# B&R Automation Studio project OPSU1
Automation Studio 4.5.2.102

## Configuration Real

### Task classes (Cpu.sw)
```
Cyclic#4:
  Main <- Main.prg
Libraries: motor
```

### Hardware
```
4PP065_0571_P74 : 4PP065.0571-P74 v1.1.2.0
  Connector IF5:
    ActivateDevice = 1
  ConfigurationID = kvbo0721lab1_Real
  Simulation = 1
```

## Logical view

Binary libraries used (declarations not repeated): operator, runtime, astime, AsIecCon

### Package Logical/Libraries - Global libraries

### Library Logical/Libraries/motor (ANSIC)

#### motor.fun - Exported functions and function blocks
```iecst
{REDUND_ERROR} {REDUND_UNREPLICABLE} FUNCTION_BLOCK FB_Motor (*TODO: Add your comment here*) (*$GROUP=User,$CAT=User,$GROUPICON=User.png,$CATICON=User.png*)
	VAR_INPUT
		u : {REDUND_UNREPLICABLE} REAL;
		phi : {REDUND_UNREPLICABLE} REAL;
		dt : {REDUND_UNREPLICABLE} REAL;
	END_VAR
	VAR_OUTPUT
		w : {REDUND_UNREPLICABLE} REAL;
	END_VAR
	VAR
		integrator : {REDUND_UNREPLICABLE} FB_Integrator;
		Tm : {REDUND_UNREPLICABLE} REAL;
		ke : {REDUND_UNREPLICABLE} REAL;
	END_VAR
END_FUNCTION_BLOCK
```

#### FB_Motor.c
```c
#include <bur/plctypes.h>
#ifdef __cplusplus
	extern "C"
	{
#endif
	#include "Library.h"
#ifdef __cplusplus
	};
#endif
/* TODO: Add your comment here */
void FB_Motor(struct FB_Motor* inst)
{
	inst->integrator.in = (inst->u*(1/inst->ke) - inst->w)*(inst->dt/inst->Tm);
	FB_integrator(&(inst->integrator));
	inst->w = inst->integrator.out;
	inst->integrator.in = inst->w*inst->dt;
	FB_integrator(&(inst->integrator));

	inst->phi = inst->integrator.out;
}
```

#### FB_Regulator.c
```c
#include <bur/plctypes.h>
#ifdef __cplusplus
	extern "C"
	{
#endif
	#include "regulator.h"
#ifdef __cplusplus
	};
#endif
/* TODO: Add your comment here */
void FB_Regulator(struct FB_Regulator* inst)
{
	inst->integrator.in = inst->e*inst->k_i*inst->dt + inst->iyOld;
	FB_integrator(&(inst->integrator));
	inst->e_p = inst->e*inst->k_p;
	if (inst->e_p < inst->max_abs_value || inst->e_p > -inst->max_abs_value);
	else
	{
		if (inst->e_p > 0) inst->e_p = inst->max_abs_value;
		else inst->e_p = -inst->max_abs_value;
	}

	inst->e_p += inst->integrator.out;
	if (inst->e_p < inst->max_abs_value || inst->e_p -inst->max_abs_value) inst->u = inst->e_p;
	else
	{
		if (inst->e_p > 0) inst->u = inst->max_abs_value;
		else inst->u = -inst->max_abs_value;
	}
	inst->iyOld = inst->u - inst->e_p;
}
```

#### FB_Integrator.c
```c
#include <bur/plctypes.h>
#ifdef __cplusplus
	extern "C"
	{
#endif
	#include "integrator.h"
#ifdef __cplusplus
	};
#endif
/* TODO: Add your comment here */
void FB_Integrator(struct FB_Integrator* inst)
{
	inst->out += inst->in;
}
```

### Program Logical/Main (ANSIC)

#### Variables.var
```iecst
VAR
	fb_controller : FB_Controller;
	fb_motor : FB_Motor;
	Enable : BOOL;
	Speed : REAL;
	fb_motor2 : FB_Motor;
	count : REAL;
	integrator : FB_Integrator;
END_VAR
```

Listed in the project but not available here: Logical/Global.typ, Logical/Global.var, Logical/Libraries/motor/Types.typ, Logical/Libraries/motor/Constants.var
